# EPICS autosave request: iocBoot/pvStatsCommon.req
$(P):INP$(N).INP
$(P):COMP$(N):100.DISA
$(P):COMP$(N):1000.DISA
$(P):COMP$(N):10000.DISA
$(P):COMP$(N):100000.DISA
$(P):INP$(N):DATAINT
$(P):INP$(N):TOTALTIME
$(P):INP$(N):USEMONITOR
$(P):INP$(N):THRESH
